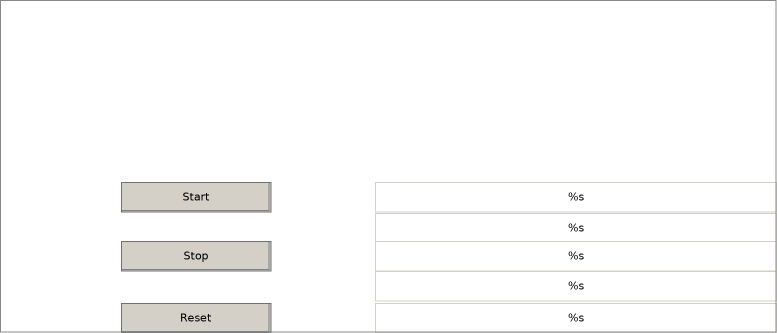
VISUALIZATION Visualization  // 777x333
    Button (121,182 150x30), "Start"
        tap GVL.Inbox_IoT_SoftStart
    Button (121,241 150x30), "Stop"
        tap GVL.Inbox_IoT_SoftStop
    Button (121,303 150x30), "Reset"
        tap GVL.Inbox_IoT_SoftReset
    Textfield (375,182 402x30), "%s", text variable: GVL.HMI_Logs[1]
    Textfield (375,213 402x30), "%s", text variable: GVL.HMI_Logs[2]
    Textfield (375,241 402x30), "%s", text variable: GVL.HMI_Logs[3]
    Textfield (375,271 402x30), "%s", text variable: GVL.HMI_Logs[4]
    Textfield (375,303 402x30), "%s", text variable: GVL.HMI_Logs[5]
END_VISUALIZATION

(* stored: Version 1.1.0.1
   Visu Visualization: Id {07edd1d1-a74f-44a5-98f6-92d028510ef9} *)
